// TIA Portal V17 export
// export: Created 2023-02-14T02:49:28.6563899Z, ExportSetting WithDefaults, DisplayName Totally Integrated Automation Portal, DisplayVersion V17, DisplayName TIA Portal Openness, DisplayVersion V17, DisplayName TIA Portal Teamcenter Gateway, DisplayVersion V17, DisplayName TIA Portal Version Control Interface, DisplayVersion V17, DisplayName SINAMICS Startdrive Advanced, DisplayVersion V17, DisplayName SINAMICS Startdrive G130, G150, S120, S150, SINAMICS MV, S210, DisplayVersion V17, DisplayName SINAMICS Startdrive G110M, G120, G120C, G120D, G120P, G115D, DisplayVersion V17, DisplayName STEP 7 Professional, DisplayVersion V17, DisplayName STEP 7 Safety, DisplayVersion V17, DisplayName WinCC Professional, DisplayVersion V17
DATA_BLOCK "IO_Valve_Blend20_DB"   // DB28
VERSION : 0.1
// stored: AutoNumber true, DBAccessibleFromOPCUA true, DBAccessibleFromWebserver true, InstanceOfName IO_Valve_Blend20, InstanceOfType FB
"IO_Valve_Blend20"
   // VAR_INPUT
   //    "lock 1" : Bool;
   //    "lock 2" : Bool;
   //    "lock 3" : Bool;
   //    "lock 4" : Bool;
   //    init : Bool;
   //    reset : Bool;
   //    testing : Bool;
   // END_VAR
   // VAR
   //    "AV-20.01" : "Valve";
   //    "AV-20.02" : "Valve";
   //    "AV-20.03" : "Valve";
   //    "AV-20.04" : "Valve";
   //    "AV-20.05" : "Valve";
   //    "AV-20.06" : "Valve";
   //    "AV-20.07" : "Valve";
   //    "AV-20.08" : "Valve";
   //    "AV-20.09" : "Valve";
   //    "AV-20.10" : "Valve";
   //    "AV-20.11" : "Valve";
   //    "AV-20.21" : "Valve";
   //    "AV-20.22" : "Valve";
   //    "AV-20.23" : "Valve";
   //    "AV-20.24" : "Valve";
   //    "AV-20.25" : "Valve";
   //    "AV-20.26" : "Valve";
   //    "AV-20.27" : "Valve";
   //    "AV-20.28" : "Valve";
   //    "AV-20.29" : "Valve";
   //    "AV-20.30" : "Valve";
   //    "AV-20.31" : "Valve";
   //    "AV-20.32" : "Valve";
   //    "AV-20.33" : "Valve";
   //    "AV-20.34" : "Valve";
   //    "AV-20.35" : "Valve";
   //    "AV-20.36" : "Valve";
   //    "AV-20.37" : "Valve";
   //    "AV-20.41" : "Valve";
   //    "AV-20.42" : "Valve";
   // END_VAR
BEGIN
END_DATA_BLOCK
